// TIA Portal V20 export
DATA_BLOCK "T5 EXCENTRIC I-O"   // DB1618
{ S7_Optimized_Access := 'TRUE' }
AUTHOR : SAS
// stored: AutoNumber false, IsRetainMemResEnabled true, MemoryReserve 100, RetainMemoryReserve 100
   VAR
      DI : Struct
         "LM5 T5-S44.5" : Bool;   // (E93.4) T5 Excentricentric Comanda 'Inainte'
         "LM5 T5-S44.6" : Bool;   // (E93.5) T5 Excentricentric Comanda 'Inapoi'
         "LM5-T5-B48.3" : Bool;   // (E97.2) T5 Excentricentric Senzor Pozitie 'Initial'
         "LM5-T5-B48.4" : Bool;   // (E97.3) T5 Excentricentric Senzor Pozitie 'Vertical'
         "TF2 T5-E102 F6.6" : Bool;   // (E170.0) T5 Excentricentric Tensiune Comanda
         "TF2 T5-E102 Q6.1" : Bool;   // (E170.1) T5 Excentricentric Disjunctor Alimentare SoftStarter SIKO
         "TF2 T5-E102 F6.1" : Bool;   // (E170.2) T5 Excentricentric Protectie Termica Motor
         "TF2 T5-E102 K6.7no" : Bool;   // (E170.3) T5 Excentricentric Confirmare Rotire 'Inainte'
         "TF2 T5-E102 K6.8no" : Bool;   // (E170.4) T5 Excentricentric Confirmare Rotire 'Inapoi'
         "TF2 T5-E102 G6.1'OK'" : Bool;   // (E170.5) T5 Excentricentric SoftStarter SIKO 'OK'
         "TF2 T5-E102 F6.3" : Bool;   // (E170.7) T5 Excentricentric Prezenta Tensiune Alimentare Frana
      END_STRUCT;
      "DO" : Struct
         "LM5-T5-H57.2" : Bool;   // (A93.1) T5 Excentric Semnalizare 'Ok'
         "LM5-T5-H57.3" : Bool;   // (A93.2) T5 Excentric Semnalizare Pozitie 'Initial'
         "TF2 T5-K53.4" : Bool;   // (A172.3) T5 Excentric Contactor Deplasare 'Inainte'
         "TF2 T5-K53.5" : Bool;   // (A172.4) T5 Excentric Contactor Deplasare 'Inapoi'
         "TF2 T5-K53.6" : Bool;   // (A172.5) T5 Excentric Contactor SoftStarter SIKO 'Start'
      END_STRUCT;
   END_VAR
BEGIN
END_DATA_BLOCK
